FUNCTION_BLOCK basicAlarmeHH_H_L_LL (* Basic Function Block Type *)
  (* Standard: 61499-2 *)
  (* Version 0.0, 1/23/2026, Schneider Electric, Template *)
  PACKAGE Hidryco.HidrycoLib;
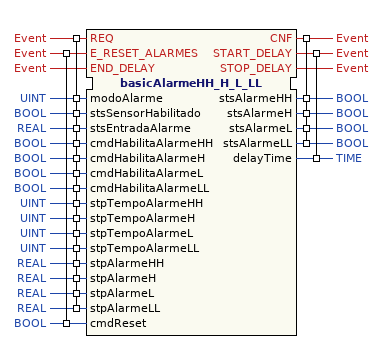
  EVENT_INPUT
    REQ WITH modoAlarme, stsSensorHabilitado, cmdHabilitaAlarmeHH, cmdHabilitaAlarmeH, cmdHabilitaAlarmeL, cmdHabilitaAlarmeLL, stpTempoAlarmeHH, stpTempoAlarmeH, stpTempoAlarmeL, stpTempoAlarmeLL, stpAlarmeHH, stpAlarmeH, stpAlarmeL, stpAlarmeLL, stsEntradaAlarme;
    E_RESET_ALARMES WITH cmdReset;
    END_DELAY;
  END_EVENT
  EVENT_OUTPUT
    CNF WITH stsAlarmeH, stsAlarmeL, stsAlarmeLL, stsAlarmeHH; (* Execution Confirmation *)
    START_DELAY WITH delayTime;
    STOP_DELAY;
  END_EVENT
  VAR_INPUT
    modoAlarme : UINT; (* Modo do alarme: 0 - AutoReset, 1 - Comando de Reset *)
    stsSensorHabilitado : BOOL;
    stsEntradaAlarme : REAL;
    cmdHabilitaAlarmeHH : BOOL;
    cmdHabilitaAlarmeH : BOOL;
    cmdHabilitaAlarmeL : BOOL;
    cmdHabilitaAlarmeLL : BOOL;
    stpTempoAlarmeHH : UINT;
    stpTempoAlarmeH : UINT;
    stpTempoAlarmeL : UINT;
    stpTempoAlarmeLL : UINT;
    stpAlarmeHH : REAL;
    stpAlarmeH : REAL;
    stpAlarmeL : REAL;
    stpAlarmeLL : REAL;
    cmdReset : BOOL;
  END_VAR
  VAR_OUTPUT
    stsAlarmeHH : BOOL; (* Output event qualifier *)
    stsAlarmeH : BOOL;
    stsAlarmeL : BOOL;
    stsAlarmeLL : BOOL;
    delayTime : TIME;
  END_VAR
  VAR
    bResetPedido : BOOL;
    bTimerExpirou : BOOL;
    bTimerAtivo : BOOL;
    iNivelTimer : INT;
    iNivelNovo : INT;
    timerCmd : INT;
    tNovo : TIME;
    bCondHH : BOOL;
    bCondH : BOOL;
    bCondL : BOOL;
    bCondLL : BOOL;
  END_VAR
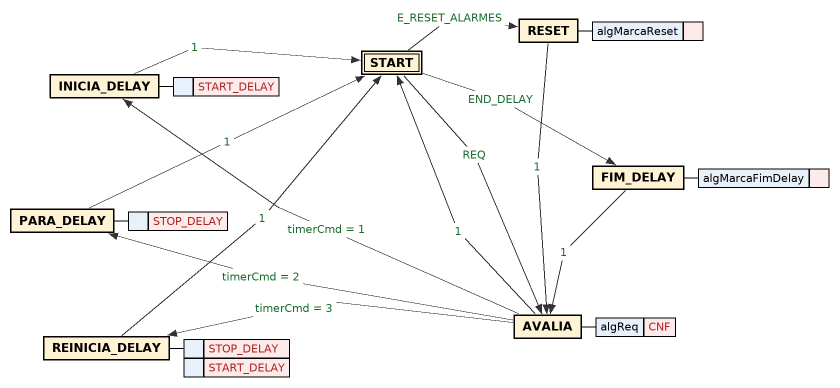
  EC_STATES
    START; (* Initial State *)
    AVALIA : algReq -> CNF;
    FIM_DELAY : algMarcaFimDelay;
    INICIA_DELAY : -> START_DELAY;
    PARA_DELAY : -> STOP_DELAY;
    REINICIA_DELAY : -> STOP_DELAY, -> START_DELAY;
    RESET : algMarcaReset;
  END_STATES
  EC_TRANSITIONS
    START TO AVALIA := REQ;
    START TO RESET := E_RESET_ALARMES;
    START TO FIM_DELAY := END_DELAY;
    RESET TO AVALIA := 1;
    FIM_DELAY TO AVALIA := 1;
    AVALIA TO PARA_DELAY := timerCmd = 2;
    AVALIA TO REINICIA_DELAY := timerCmd = 3;
    AVALIA TO INICIA_DELAY := timerCmd = 1;
    AVALIA TO START := 1;
    INICIA_DELAY TO START := 1;
    PARA_DELAY TO START := 1;
    REINICIA_DELAY TO START := 1;
  END_TRANSITIONS
  ALGORITHM algMarcaFimDelay IN ST:
bTimerExpirou := bTimerAtivo;
;
  END_ALGORITHM
  ALGORITHM algReq IN ST:
timerCmd := 0;

(* ---- Sensor desabilitado: zera tudo ---- *)
IF NOT stsSensorHabilitado THEN
    stsAlarmeHH := FALSE;
    stsAlarmeH  := FALSE;
    stsAlarmeL  := FALSE;
    stsAlarmeLL := FALSE;
    bResetPedido  := FALSE;
    bTimerExpirou := FALSE;
    IF bTimerAtivo THEN
        timerCmd := 2;
    END_IF;
    bTimerAtivo := FALSE;
    iNivelTimer := 0;
    RETURN;
END_IF;

(* ---- Condições atuais ---- *)
bCondHH := cmdHabilitaAlarmeHH AND (stsEntradaAlarme > stpAlarmeHH);
bCondH  := cmdHabilitaAlarmeH  AND (stsEntradaAlarme > stpAlarmeH);
bCondL  := cmdHabilitaAlarmeL  AND (stsEntradaAlarme < stpAlarmeL);
bCondLL := cmdHabilitaAlarmeLL AND (stsEntradaAlarme < stpAlarmeLL);

(* ---- Alarme desabilitado zera o próprio alarme ---- *)
IF NOT cmdHabilitaAlarmeHH THEN stsAlarmeHH := FALSE; END_IF;
IF NOT cmdHabilitaAlarmeH  THEN stsAlarmeH  := FALSE; END_IF;
IF NOT cmdHabilitaAlarmeL  THEN stsAlarmeL  := FALSE; END_IF;
IF NOT cmdHabilitaAlarmeLL THEN stsAlarmeLL := FALSE; END_IF;

(* ---- Tempo esgotado: ativa todos cuja condição persiste ---- *)
IF bTimerExpirou THEN
    IF bCondHH THEN stsAlarmeHH := TRUE; END_IF;
    IF bCondH  THEN stsAlarmeH  := TRUE; END_IF;
    IF bCondL  THEN stsAlarmeL  := TRUE; END_IF;
    IF bCondLL THEN stsAlarmeLL := TRUE; END_IF;
    bTimerExpirou := FALSE;
    bTimerAtivo   := FALSE;
    iNivelTimer   := 0;
END_IF;

(* ---- Reset ---- *)
IF modoAlarme = 0 THEN
    (* automático, histerese de 10% do setpoint *)
    IF stsAlarmeHH AND (stsEntradaAlarme <= stpAlarmeHH - ABS(stpAlarmeHH) * 0.1) THEN stsAlarmeHH := FALSE; END_IF;
    IF stsAlarmeH  AND (stsEntradaAlarme <= stpAlarmeH  - ABS(stpAlarmeH)  * 0.1) THEN stsAlarmeH  := FALSE; END_IF;
    IF stsAlarmeL  AND (stsEntradaAlarme >= stpAlarmeL  + ABS(stpAlarmeL)  * 0.1) THEN stsAlarmeL  := FALSE; END_IF;
    IF stsAlarmeLL AND (stsEntradaAlarme >= stpAlarmeLL + ABS(stpAlarmeLL) * 0.1) THEN stsAlarmeLL := FALSE; END_IF;
ELSIF bResetPedido THEN
    (* manual, sem histerese: só zera se o valor já voltou *)
    IF stsAlarmeHH AND (stsEntradaAlarme <= stpAlarmeHH) THEN stsAlarmeHH := FALSE; END_IF;
    IF stsAlarmeH  AND (stsEntradaAlarme <= stpAlarmeH)  THEN stsAlarmeH  := FALSE; END_IF;
    IF stsAlarmeL  AND (stsEntradaAlarme >= stpAlarmeL)  THEN stsAlarmeL  := FALSE; END_IF;
    IF stsAlarmeLL AND (stsEntradaAlarme >= stpAlarmeLL) THEN stsAlarmeLL := FALSE; END_IF;
END_IF;
bResetPedido := FALSE;

(* ---- Pendente de maior prioridade (HH > H > LL > L) ---- *)
iNivelNovo := 0;
IF bCondHH AND NOT stsAlarmeHH THEN
    iNivelNovo := 1; tNovo := DINT_TO_TIME(UINT_TO_DINT(stpTempoAlarmeHH) * 1000);
ELSIF bCondH AND NOT stsAlarmeH THEN
    iNivelNovo := 2; tNovo := DINT_TO_TIME(UINT_TO_DINT(stpTempoAlarmeH) * 1000);
ELSIF bCondLL AND NOT stsAlarmeLL THEN
    iNivelNovo := 3; tNovo := DINT_TO_TIME(UINT_TO_DINT(stpTempoAlarmeLL) * 1000);
ELSIF bCondL AND NOT stsAlarmeL THEN
    iNivelNovo := 4; tNovo := DINT_TO_TIME(UINT_TO_DINT(stpTempoAlarmeL) * 1000);
END_IF;

(* ---- Decisão do temporizador ---- *)
IF iNivelNovo = 0 THEN
    IF bTimerAtivo THEN
        timerCmd := 2;                  (* condição sumiu: cancela *)
    END_IF;
    bTimerAtivo := FALSE;
    iNivelTimer := 0;
ELSIF NOT bTimerAtivo THEN
    delayTime   := tNovo;
    timerCmd    := 1;                   (* inicia *)
    bTimerAtivo := TRUE;
    iNivelTimer := iNivelNovo;
ELSIF iNivelNovo <> iNivelTimer THEN
    delayTime   := tNovo;
    timerCmd    := 3;                   (* troca de nível: reinicia com o novo tempo *)
    iNivelTimer := iNivelNovo;
END_IF;
;
  END_ALGORITHM
  ALGORITHM algMarcaReset IN ST:
bResetPedido := cmdReset;
;
  END_ALGORITHM
END_FUNCTION_BLOCK
